// TIA Portal V19 export
FUNCTION "Ergebnis_DT" : Void   // FC340, LAD
TITLE = Ergebnis speichern
{ S7_Optimized_Access := 'TRUE' }
// stored: AutoNumber false, SetENOAutomatically false
   VAR_INPUT
      "Name" : String;
      akt_Zeit : DTL;
      ok : Bool;
      Fehler : Bool;
   END_VAR
   VAR_TEMP
      i : Int;
   END_VAR
BEGIN

REGION Network 1 (SCL)
   //Index erhöhen
   "Drucktest".akt_Index := "Drucktest".akt_Index + 1;
   IF "Drucktest".akt_Index > 100 THEN
       "Drucktest".akt_Index := 1;
   END_IF;
   #i := "Drucktest".akt_Index;
   // --> Speichern
   "Drucktest".Ergebnis[#i].Name := #Name;

   "Drucktest".Ergebnis[#i].Zeit := #akt_Zeit;

   "Drucktest".Ergebnis[#i].ok := #ok;

   "Drucktest".Ergebnis[#i].Fehler := #Fehler;
END_REGION
END_FUNCTION
